FUNCTION alg_a_x: BOOL
{ S7_Optimized_Access := 'false' }
    VAR_INPUT
        state: STATE;
    END_VAR

BEGIN
    alg_a_x := TRUE;
END_FUNCTION
